Staubli VAL3: goHome.pgx

program goHome()
begin
  if !bHome
    resetMotion()
    pCurrent=here(date:tTCP,date:fWorkTable)
    //判断是否在打磨区域
    if pCurrent.trsf.z<100
      movel(appro(pCurrent,{0,0,-50,0,0,0}),date:tTCP,date:mNomSpeed)
    endIf
    movej(date:jHome,date:tTCP,date:mNomSpeed)
    waitEndMove()
    call massage("到达零位")
  endIf

end
